// TIA Portal V17 export
// export: Created 2024-08-20T11:47:11.8553107Z, ExportSetting WithDefaults, DisplayName Totally Integrated Automation Portal, DisplayVersion V17 Update 4, DisplayName TIA Portal Openness, DisplayVersion V17 Update 4, DisplayName TIA Portal Version Control Interface, DisplayVersion V17, DisplayName STEP 7 Professional, DisplayVersion V17 Update 4, DisplayName STEP 7 Safety, DisplayVersion V17, DisplayName WinCC Advanced, DisplayVersion V17 Update 4
FUNCTION_BLOCK "teste"   // FB1, SCL
{ S7_Optimized_Access := 'TRUE' }
VERSION : 0.1
// stored: AutoNumber true, IsIECCheckEnabled false, IsRetainMemResEnabled false, MemoryReserve 100, SetENOAutomatically false, UDAEnableTagReadback false
   VAR
      tag1 : Int;
      tag2 : Int;
      tag3 : Int;
   END_VAR
BEGIN

   #tag1 := 0;


   WHILE #tag1 < 100 DO
       #tag1 := #tag1 + 1;
           IF #tag1 >= 99 THEN
               #tag1 := 0;
           END_IF;// Statement section WHILE
   END_WHILE;
END_FUNCTION_BLOCK
